// SIMATIC S7-200 project (STEP 7-Micro/WIN), CPU 221 REL 01.10

ORGANIZATION_BLOCK 主程序:OB1
TITLE=程序注释
BEGIN
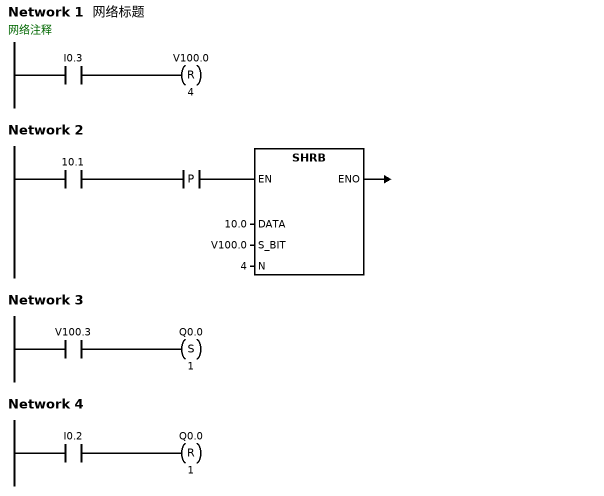
Network 1 // 网络标题
// 网络注释
// (network saved uncompiled; LAD cells follow)
// row 0: c0 -| |- I0.3  c1 -(R) V100.0, 4
Network 2
// (network saved uncompiled; LAD cells follow)
// row 0: c0 -| |- 10.1  c1 -|P|-  c2 [SHRB EN:=power@row0, DATA:=10.0, S_BIT:=V100.0, N:=4, ENO=>power]  c3 ->
// row 1: c2 [box]
Network 3
LD     V100.3
S      Q0.0, 1
Network 4
LD     I0.2
R      Q0.0, 1
END_ORGANIZATION_BLOCK
